TYPE Layer :
STRUCT
	num_neurons : UINT;
	activation : act_type;
	pointer_weight: POINTER TO LREAL;
	pointer_bias: POINTER TO LREAL;
	normalization: act_type;
END_STRUCT
END_TYPE

(* stored: Version 1.1.0.1, ProductVersion 3.1.4024.12
   DUT Layer: Id {fd28c200-5075-457e-a386-302b613d5a8f} *)
